FUNCTION_BLOCK SET_STRUCT_VALUE (* Service Interface Function Block Type *)
  PACKAGE eclipse4diac::convert;
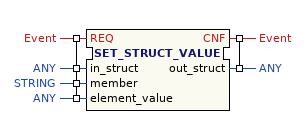
  EVENT_INPUT
    REQ WITH member, in_struct, element_value; (* Set Value out of structure *)
  END_EVENT
  EVENT_OUTPUT
    CNF WITH out_struct; (* REQ event finished *)
  END_EVENT
  VAR_INPUT
    in_struct : ANY; (* Structure to look into *)
    member : STRING; (* Member of the strucuture to retrieve. Inner members are access using the dot (.) operator *)
    element_value : ANY; (* new value for the element *)
  END_VAR
  VAR_OUTPUT
    out_struct : ANY; (* TRUE if no errors ocurred, FALSE otherwise *)
  END_VAR
END_FUNCTION_BLOCK
